{attribute 'qualified_only'}
VAR_GLOBAL
	_MotorOnOff				:BOOL;
	_SensorCovered			:BOOL;
	_Switch					:BOOL;
	_PackageIsPlaced		:BOOL;
	_RetainedTimeOnConveyor	:TIME;
	_MovementTime			:TIME := T#10S;		//How long it takes for the package to move through the conveyor
END_VAR

(* stored: Version 1.1.0.1
   GVL GVL: Id {723f8d7e-b51b-45f9-a87d-77ccdd2fd663} *)
